Fanuc KAREL source: kd00045.KL

-- PROVISIONAL review KL for V770-1; original PC SHA256 ea9ff8bdccfbc1d8eca07d0589d1a72ccfb41312f2796ef77c716e2af386bb4a
-- Incomplete behavior may be omitted. Consult companion uncertainty JSON. Do not deploy.
PROGRAM KD00045
%NOLOCKGROUP
VAR
  I : INTEGER
  J : INTEGER
  B : BOOLEAN
  R : REAL
  S : STRING[80]
-- UNRESOLVED_DECL P type=000101
BEGIN
  -- UNRESOLVED_PC offsets 5-24; opcodes 01,22,1C,06,82,0B
  -- UNRESOLVED_PC offsets 29-33; opcodes 7F
END KD00045
